// TIA Portal V20 export
DATA_BLOCK "InstShiftmodel"   // DB101
TITLE = Instanz Shiftmodel / InstanceShiftmodel
{ DB_Accessible_From_OPC_UA := 'FALSE' }
AUTHOR : SICAR
FAMILY : Shiftmodel
// Instanz DB / Instance DB
// stored: DBAccessibleFromOPCUA false, InstanceOfName LSicar_Shiftmodel, InstanceOfType FB
"LSicar_Shiftmodel"
   // VAR_OUTPUT
   //    currentShiftCircuitTimes { ExternalAccessible := 'False'; ExternalVisible := 'False'; ExternalWritable := 'False'} : "LSicar_typeShiftmodTime1Shift";
   //    currentShiftTimes { ExternalAccessible := 'False'; ExternalVisible := 'False'; ExternalWritable := 'False'} : "LSicar_typeShiftTimes1Shift";
   // END_VAR
   // VAR_IN_OUT
   //    dateAndTime : "LSicar_typeGlobalDateTime";
   //    shiftTimesHmi : "LSicar_typeShiftmodelHmi";
   //    shiftTimesList : Array[0..10] of "LSicar_typeShiftmodTime1DaySel";
   // END_VAR
   // VAR
   //    statListIdx { ExternalAccessible := 'False'; ExternalVisible := 'False'; ExternalWritable := 'False'} : DInt;
   //    statHmiTimesDay { ExternalAccessible := 'False'; ExternalVisible := 'False'; ExternalWritable := 'False'} : Array[0..7] of "LSicar_typeShiftmodTime1Day";
   //    statHmiSignalsDay { ExternalAccessible := 'False'; ExternalVisible := 'False'; ExternalWritable := 'False'} : Array[0..7] of "LSicar_typeShiftmodSign1Day";
   //    statHmiActualDay { ExternalAccessible := 'False'; ExternalVisible := 'False'; ExternalWritable := 'False'} : USInt;
   //    statShiftTimesListOn { ExternalAccessible := 'False'; ExternalVisible := 'False'; ExternalWritable := 'False'} : Bool;
   //    statSummaryHmi { ExternalAccessible := 'False'; ExternalVisible := 'False'; ExternalWritable := 'False'} : "LSicar_typeShiftmodSumHmi";
   //    statHmiShiftmoListindex { ExternalAccessible := 'False'; ExternalVisible := 'False'; ExternalWritable := 'False'} : USInt;
   //    statZeroDay { ExternalAccessible := 'False'; ExternalVisible := 'False'; ExternalWritable := 'False'} : "LSicar_typeShiftmodTime1Day";
   //    statListIndexOld { ExternalAccessible := 'False'; ExternalVisible := 'False'; ExternalWritable := 'False'} : DInt;
   //    statNumberOfWorkDays { ExternalAccessible := 'False'; ExternalVisible := 'False'; ExternalWritable := 'False'} : USInt;
   //    statTimeOfDayActual { ExternalAccessible := 'False'; ExternalVisible := 'False'; ExternalWritable := 'False'} : Time_Of_Day;
   //    statShiftActual { ExternalAccessible := 'False'; ExternalVisible := 'False'; ExternalWritable := 'False'} : USInt;
   //    statDayCount { ExternalAccessible := 'False'; ExternalVisible := 'False'; ExternalWritable := 'False'} : USInt;
   //    statBreakCount { ExternalAccessible := 'False'; ExternalVisible := 'False'; ExternalWritable := 'False'} : USInt;
   //    statDayChangeNightShift { ExternalAccessible := 'False'; ExternalVisible := 'False'; ExternalWritable := 'False'} : Bool;
   //    statDayChangeCircuitTime { ExternalAccessible := 'False'; ExternalVisible := 'False'; ExternalWritable := 'False'} : Bool;
   //    statCheckCircuitTime { ExternalAccessible := 'False'; ExternalVisible := 'False'; ExternalWritable := 'False'} : "LSicar_typeShiftCircuitTimes";
   //    statRisEdge { ExternalAccessible := 'False'; ExternalVisible := 'False'; ExternalWritable := 'False'} : "LSicar_typeShiftmodSumHmi";
   //    statPosPulse { ExternalAccessible := 'False'; ExternalVisible := 'False'; ExternalWritable := 'False'} : "LSicar_typeShiftmodSumHmi";
   //    statFalEdge { ExternalAccessible := 'False'; ExternalVisible := 'False'; ExternalWritable := 'False'} : "LSicar_typeShiftmodSumHmi";
   //    statNegPulse { ExternalAccessible := 'False'; ExternalVisible := 'False'; ExternalWritable := 'False'} : "LSicar_typeShiftmodSumHmi";
   //    statTimesAndCircuit { ExternalAccessible := 'False'; ExternalVisible := 'False'; ExternalWritable := 'False'} : "LSicar_typeShiftmodTime1Shift";
   //    statOnlyTimes { ExternalAccessible := 'False'; ExternalVisible := 'False'; ExternalWritable := 'False'} : "LSicar_typeShiftTimes1Shift";
   //    statRisEdgeListOn { ExternalAccessible := 'False'; ExternalVisible := 'False'; ExternalWritable := 'False'} : Bool;
   //    statPosPulseListOn { ExternalAccessible := 'False'; ExternalVisible := 'False'; ExternalWritable := 'False'} : Bool;
   //    statFalEdgeListOn { ExternalAccessible := 'False'; ExternalVisible := 'False'; ExternalWritable := 'False'} : Bool;
   //    statNegPulseListOn { ExternalAccessible := 'False'; ExternalVisible := 'False'; ExternalWritable := 'False'} : Bool;
   //    statRisEdgeListChange { ExternalAccessible := 'False'; ExternalVisible := 'False'; ExternalWritable := 'False'} : Bool;
   //    statPosPulseListChange { ExternalAccessible := 'False'; ExternalVisible := 'False'; ExternalWritable := 'False'} : Bool;
   //    statFirstCycle { ExternalAccessible := 'False'; ExternalVisible := 'False'; ExternalWritable := 'False'} : Bool;
   // END_VAR
BEGIN
END_DATA_BLOCK
